                // Counter delta with 32-bit wrap support.
                // This also allows negative movement when converted to DINT.
                counterDeltaCh1 := UDINT_TO_DINT(encoderPositionRawValue - lastCounterValueCh1);

                // Convert pulses to millimeters
                positionDeltaCh1 := DINT_TO_REAL(counterDeltaCh1) * encoderScalingFactor;

                // Calculate speed
                channel1EncoderSpeedMMs := positionDeltaCh1 / calculationTimeSec;
                channel1EncoderSpeedMPM := channel1EncoderSpeedMMs * 60.0 / 1000.0;

                // Absolute speed
                channel1EncoderSpeedAbsMMs := ABS(channel1EncoderSpeedMMs);
                channel1EncoderSpeedAbsMPM := ABS(channel1EncoderSpeedMPM);

            ELSE
                // First cycle has no valid previous counter
                channel1EncoderSpeedMMs    := 0.0;
                channel1EncoderSpeedMPM    := 0.0;
                channel1EncoderSpeedAbsMMs := 0.0;
                channel1EncoderSpeedAbsMPM := 0.0;

                firstCycleCh1 := FALSE;
            END_IF

            // Store current counter for next calculation
            lastCounterValueCh1 := encoderPositionRawValue;
        END_IF


    //==============================================================
    // CHANNEL 2
    //==============================================================
    2:
        instTON_calculateEncSpeedCh2(IN := TRUE, PT := speedCalculationCycleTime);

        IF instTON_calculateEncSpeedCh2.Q THEN
            // Reset timer
            instTON_calculateEncSpeedCh2(IN := FALSE);

            IF NOT firstCycleCh2 THEN

                // Counter delta with 32-bit wrap support.
                // This also allows negative movement when converted to DINT.
                counterDeltaCh2 := UDINT_TO_DINT(encoderPositionRawValue - lastCounterValueCh2);

                // Convert pulses to millimeters
                positionDeltaCh2 := DINT_TO_REAL(counterDeltaCh2) * encoderScalingFactor;

                // Calculate speed
                channel2EncoderSpeedMMs := positionDeltaCh2 / calculationTimeSec;
                channel2EncoderSpeedMPM := channel2EncoderSpeedMMs * 60.0 / 1000.0;

                // Absolute speed
                channel2EncoderSpeedAbsMMs := ABS(channel2EncoderSpeedMMs);
                channel2EncoderSpeedAbsMPM := ABS(channel2EncoderSpeedMPM);

            ELSE
                // First cycle has no valid previous counter
                channel2EncoderSpeedMMs    := 0.0;
                channel2EncoderSpeedMPM    := 0.0;
                channel2EncoderSpeedAbsMMs := 0.0;
                channel2EncoderSpeedAbsMPM := 0.0;

                firstCycleCh2 := FALSE;
            END_IF

            // Store current counter for next calculation
            lastCounterValueCh2 := encoderPositionRawValue;
        END_IF

END_CASE
END_METHOD

METHOD PRIVATE _CalculateModuloPosition : LREAL
// ==================================================================================================
// Calculates modulo position without using FLOOR.
//
// Output range:
//   0.0 <= modulo position < moduloPosition
//
// Example:
//   absolutePosition = 725.0
//   moduloPosition   = 360.0
//   return           = 5.0
// ==================================================================================================

VAR_INPUT
    absolutePosition : LREAL; // Absolute accumulated position
    moduloPosition   : LREAL; // Modulo range, for example 360.0
END_VAR

VAR
    quotient    : LINT;
    moduloValue : LREAL;
END_VAR


// If modulo is disabled or invalid, return absolute position
IF moduloPosition <= 0.0 THEN
    _CalculateModuloPosition := absolutePosition;
    RETURN;
END_IF


// Approximate quotient.
// Depending on the PLC/runtime, LREAL_TO_LINT may truncate or round.
// The correction below guarantees the final value stays inside the modulo range.
quotient := LREAL_TO_LINT(absolutePosition / moduloPosition);


// Calculate initial modulo value
moduloValue := absolutePosition - (LINT_TO_LREAL(quotient) * moduloPosition);


// Correct negative residue
WHILE moduloValue < 0.0 DO
    moduloValue := moduloValue + moduloPosition;
END_WHILE


// Correct value above modulo range
WHILE moduloValue >= moduloPosition DO
    moduloValue := moduloValue - moduloPosition;
END_WHILE


_CalculateModuloPosition := moduloValue;
END_METHOD

METHOD PRIVATE _SetEncoderPosition
// ==================================================================================================
// Sets encoder position for channel 1 or channel 2.
//
// The command is triggered on the rising edge of setPosition.
// The desired position in millimeters is converted to raw encoder pulses.
// ==================================================================================================

VAR_INPUT
    channel              : USINT; // 1 = Channel 1, 2 = Channel 2
    setPosition          : BOOL;  // Rising edge command
    desiredPosition      : LREAL; // Desired position in mm
    encoderScalingFactor : REAL;  // mm per pulse
END_VAR

VAR
    setPositionRawValue : UDINT;
END_VAR


IF encoderScalingFactor <= 0.0 THEN
    RETURN;
END_IF


// Convert desired position from mm to raw encoder pulses
setPositionRawValue := LREAL_TO_UDINT(desiredPosition / REAL_TO_LREAL(encoderScalingFactor));


CASE channel OF

    //==============================================================
    // CHANNEL 1
    //==============================================================
    1:

        // Rising edge detection
        IF setPosition AND NOT channel1SetPositionOld THEN

            channel1SetPositionRawValue := setPositionRawValue;

            // Write raw set value to output PDO
            // Adjust these member names according to your EL5152_PLCTOHW structure
            PlcToHw.channel1.setCounterValue := channel1SetPositionRawValue;

            // Generate one PLC-cycle command pulse
            // Adjust this member name according to your EL5152_PLCTOHW structure
            PlcToHw.channel1.control.Set_counter := TRUE;

            // Avoid false speed spike after position jump
            firstCycleCh1 := TRUE;

        ELSE

            // Reset command bit after one PLC cycle
            // Adjust this member name according to your EL5152_PLCTOHW structure
            PlcToHw.channel1.control.Set_counter := FALSE;

        END_IF

        channel1SetPositionOld := setPosition;


    //==============================================================
    // CHANNEL 2
    //==============================================================
    2:

        // Rising edge detection
        IF setPosition AND NOT channel2SetPositionOld THEN

            channel2SetPositionRawValue := setPositionRawValue;

            // Write raw set value to output PDO
            // Adjust these member names according to your EL5152_PLCTOHW structure
            PlcToHw.channel2.setCounterValue := channel2SetPositionRawValue;

            // Generate one PLC-cycle command pulse
            // Adjust this member name according to your EL5152_PLCTOHW structure
            PlcToHw.channel2.control.Set_counter := TRUE;

            // Avoid false speed spike after position jump
            firstCycleCh2 := TRUE;

        ELSE

            // Reset command bit after one PLC cycle
            // Adjust this member name according to your EL5152_PLCTOHW structure
            PlcToHw.channel2.control.Set_counter := FALSE;

        END_IF

        channel2SetPositionOld := setPosition;

END_CASE
END_METHOD

METHOD PRIVATE _SimulateEncoderSpeed : UDINT
// ==================================================================================================
// Simulates encoder motion by incrementing a virtual counter value based on a given speed in m/min.
//
// Positive simulateSpeedMPM increases the raw counter.
// Negative simulateSpeedMPM decreases the raw counter.
// ==================================================================================================

VAR_INPUT
    channel              : USINT; // 1 = Channel 1, 2 = Channel 2
    encoderScalingFactor : REAL;  // Encoder resolution: mm per pulse
    simulateSpeedMPM     : REAL;  // Target speed in meters per minute
END_VAR


IF encoderScalingFactor <= 0.0 THEN
    RETURN;
END_IF


CASE channel OF

    //==============================================================
    // CHANNEL 1
    //==============================================================
    1:
        currentSystemTimeCh1 := F_GetSystemTime();

        // Initialize simulation time reference
        IF NOT simulationInitCh1 THEN
            lastCycleTimeCh1 := currentSystemTimeCh1;
            simulationInitCh1 := TRUE;
            _SimulateEncoderSpeed := simulatedPositionRawValueCh1;
            RETURN;
        END_IF

        // 1 tick = 100 ns
        // 1 ms = 10,000 ticks
        deltaTimeMsCh1 := ULINT_TO_REAL(currentSystemTimeCh1 - lastCycleTimeCh1) / 10000.0;

        // Store time for next cycle
        lastCycleTimeCh1 := currentSystemTimeCh1;

        IF deltaTimeMsCh1 > 0.0 THEN

            // Convert m/min to pulses per second
            pulsesPerSecondCh1 := (simulateSpeedMPM * 1000.0 / 60.0) / encoderScalingFactor;

            // Convert pulses per second to pulses per cycle
            pulsesToAddCh1 := REAL_TO_DINT(pulsesPerSecondCh1 * (deltaTimeMsCh1 / 1000.0));

            IF pulsesToAddCh1 >= 0 THEN
                simulatedPositionRawValueCh1 := simulatedPositionRawValueCh1 + DINT_TO_UDINT(pulsesToAddCh1);
            ELSE
                simulatedPositionRawValueCh1 := simulatedPositionRawValueCh1 - DINT_TO_UDINT(ABS(pulsesToAddCh1));
            END_IF

        END_IF

        _SimulateEncoderSpeed := simulatedPositionRawValueCh1;


    //==============================================================
    // CHANNEL 2
    //==============================================================
    2:
        currentSystemTimeCh2 := F_GetSystemTime();

        // Initialize simulation time reference
        IF NOT simulationInitCh2 THEN
            lastCycleTimeCh2 := currentSystemTimeCh2;
            simulationInitCh2 := TRUE;
            _SimulateEncoderSpeed := simulatedPositionRawValueCh2;
            RETURN;
        END_IF

        // 1 tick = 100 ns
        // 1 ms = 10,000 ticks
        deltaTimeMsCh2 := ULINT_TO_REAL(currentSystemTimeCh2 - lastCycleTimeCh2) / 10000.0;

        // Store time for next cycle
        lastCycleTimeCh2 := currentSystemTimeCh2;

        IF deltaTimeMsCh2 > 0.0 THEN

            // Convert m/min to pulses per second
            pulsesPerSecondCh2 := (simulateSpeedMPM * 1000.0 / 60.0) / encoderScalingFactor;

            // Convert pulses per second to pulses per cycle
            pulsesToAddCh2 := REAL_TO_DINT(pulsesPerSecondCh2 * (deltaTimeMsCh2 / 1000.0));

            IF pulsesToAddCh2 >= 0 THEN
                simulatedPositionRawValueCh2 := simulatedPositionRawValueCh2 + DINT_TO_UDINT(pulsesToAddCh2);
            ELSE
                simulatedPositionRawValueCh2 := simulatedPositionRawValueCh2 - DINT_TO_UDINT(ABS(pulsesToAddCh2));
            END_IF

        END_IF

        _SimulateEncoderSpeed := simulatedPositionRawValueCh2;

END_CASE
END_METHOD

END_FUNCTION_BLOCK

// ---- Library/FAS/IO-Link/006B51 - IO-Link Master/_FB_006B51.TcPOU
FUNCTION_BLOCK _FB_006B51
VAR_INPUT
	
		
END_VAR
VAR_OUTPUT
	
	channel_0 : _006B51_Channel_State;
	channel_1 : _006B51_Channel_State;
	channel_2 : _006B51_Channel_State;
	channel_3 : _006B51_Channel_State;
	channel_4 : _006B51_Channel_State;
	channel_5 : _006B51_Channel_State;
	channel_6 : _006B51_Channel_State;
	channel_7 : _006B51_Channel_State;
	
	HwToPlc	AT %I* 	: _006B51_HWTOPLC_PDOS;	
			
END_VAR

//============================================================
// CHANNEL 0
//============================================================
channel_0.inputPin2   := HwToPlc.inputPin2.00;
channel_0.inputPin4   := HwToPlc.inputPin4.00;
channel_0.deviceState := HwToPlc.deviceState.00;

// Reset port mode states
channel_0.state_PortInNoDigitalInput        := FALSE;
channel_0.state_PortInNcDigitalInput        := FALSE;
channel_0.state_PortInDigitalOutput         := FALSE;
channel_0.state_PortInIoLink                := FALSE;

// Reset diagnostic / communication states
channel_0.state_NoDeviceDetected            := FALSE;
channel_0.state_IoLinkCommunicationStatus   := FALSE;
channel_0.state_InvalidVendorId             := FALSE;
channel_0.state_InvalidDeviceId             := FALSE;
channel_0.state_InvalidSerialNumber         := FALSE;
channel_0.state_InvalidCycleTime            := FALSE;
channel_0.state_InvalidProcessDataInLength  := FALSE;
channel_0.state_InvalidProcessDataOutLength := FALSE;
channel_0.state_InvalidIoLinkVersion        := FALSE;

// Low nibble = port mode
CASE (HwToPlc.ioLinkDeviceState_Port0 AND 16#0F) OF
    16#0: channel_0.state_PortInNoDigitalInput := TRUE;
    16#1: channel_0.state_PortInNcDigitalInput := TRUE;
    16#2: channel_0.state_PortInDigitalOutput  := TRUE;
    16#3: channel_0.state_PortInIoLink         := TRUE;
END_CASE;

// High nibble = diagnostic / communication state
CASE SHR((HwToPlc.ioLinkDeviceState_Port0 AND 16#F0), 4) OF
    16#0: channel_0.state_NoDeviceDetected            := TRUE;
    16#1: channel_0.state_IoLinkCommunicationStatus   := TRUE;
    16#2: channel_0.state_InvalidVendorId             := TRUE;
    16#3: channel_0.state_InvalidDeviceId             := TRUE;
    16#4: channel_0.state_InvalidSerialNumber         := TRUE;
    16#8: channel_0.state_InvalidCycleTime            := TRUE;
    16#9: channel_0.state_InvalidProcessDataInLength  := TRUE;
    16#A: channel_0.state_InvalidProcessDataOutLength := TRUE;
    16#C: channel_0.state_InvalidIoLinkVersion        := TRUE;
END_CASE;


//============================================================
// CHANNEL 1
//============================================================
channel_1.inputPin2   := HwToPlc.inputPin2.01;
channel_1.inputPin4   := HwToPlc.inputPin4.01;
channel_1.deviceState := HwToPlc.deviceState.01;

// Reset port mode states
channel_1.state_PortInNoDigitalInput        := FALSE;
channel_1.state_PortInNcDigitalInput        := FALSE;
channel_1.state_PortInDigitalOutput         := FALSE;
channel_1.state_PortInIoLink                := FALSE;

// Reset diagnostic / communication states
channel_1.state_NoDeviceDetected            := FALSE;
channel_1.state_IoLinkCommunicationStatus   := FALSE;
channel_1.state_InvalidVendorId             := FALSE;
channel_1.state_InvalidDeviceId             := FALSE;
channel_1.state_InvalidSerialNumber         := FALSE;
channel_1.state_InvalidCycleTime            := FALSE;
channel_1.state_InvalidProcessDataInLength  := FALSE;
channel_1.state_InvalidProcessDataOutLength := FALSE;
channel_1.state_InvalidIoLinkVersion        := FALSE;

// Low nibble = port mode
CASE (HwToPlc.ioLinkDeviceState_Port1 AND 16#0F) OF
    16#0: channel_1.state_PortInNoDigitalInput := TRUE;
    16#1: channel_1.state_PortInNcDigitalInput := TRUE;
    16#2: channel_1.state_PortInDigitalOutput  := TRUE;
    16#3: channel_1.state_PortInIoLink         := TRUE;
END_CASE;

// High nibble = diagnostic / communication state
CASE SHR((HwToPlc.ioLinkDeviceState_Port1 AND 16#F0), 4) OF
    16#0: channel_1.state_NoDeviceDetected            := TRUE;
    16#1: channel_1.state_IoLinkCommunicationStatus   := TRUE;
    16#2: channel_1.state_InvalidVendorId             := TRUE;
    16#3: channel_1.state_InvalidDeviceId             := TRUE;
    16#4: channel_1.state_InvalidSerialNumber         := TRUE;
    16#8: channel_1.state_InvalidCycleTime            := TRUE;
    16#9: channel_1.state_InvalidProcessDataInLength  := TRUE;
    16#A: channel_1.state_InvalidProcessDataOutLength := TRUE;
    16#C: channel_1.state_InvalidIoLinkVersion        := TRUE;
END_CASE;


//============================================================
// CHANNEL 2
//============================================================
channel_2.inputPin2   := HwToPlc.inputPin2.02;
channel_2.inputPin4   := HwToPlc.inputPin4.02;
channel_2.deviceState := HwToPlc.deviceState.02;

// Reset port mode states
channel_2.state_PortInNoDigitalInput        := FALSE;
channel_2.state_PortInNcDigitalInput        := FALSE;
channel_2.state_PortInDigitalOutput         := FALSE;
channel_2.state_PortInIoLink                := FALSE;

// Reset diagnostic / communication states
channel_2.state_NoDeviceDetected            := FALSE;
channel_2.state_IoLinkCommunicationStatus   := FALSE;
channel_2.state_InvalidVendorId             := FALSE;
channel_2.state_InvalidDeviceId             := FALSE;
channel_2.state_InvalidSerialNumber         := FALSE;
channel_2.state_InvalidCycleTime            := FALSE;
channel_2.state_InvalidProcessDataInLength  := FALSE;
channel_2.state_InvalidProcessDataOutLength := FALSE;
channel_2.state_InvalidIoLinkVersion        := FALSE;

// Low nibble = port mode
CASE (HwToPlc.ioLinkDeviceState_Port2 AND 16#0F) OF
    16#0: channel_2.state_PortInNoDigitalInput := TRUE;
    16#1: channel_2.state_PortInNcDigitalInput := TRUE;
    16#2: channel_2.state_PortInDigitalOutput  := TRUE;
    16#3: channel_2.state_PortInIoLink         := TRUE;
END_CASE;

// High nibble = diagnostic / communication state
CASE SHR((HwToPlc.ioLinkDeviceState_Port2 AND 16#F0), 4) OF
    16#0: channel_2.state_NoDeviceDetected            := TRUE;
    16#1: channel_2.state_IoLinkCommunicationStatus   := TRUE;
    16#2: channel_2.state_InvalidVendorId             := TRUE;
    16#3: channel_2.state_InvalidDeviceId             := TRUE;
    16#4: channel_2.state_InvalidSerialNumber         := TRUE;
    16#8: channel_2.state_InvalidCycleTime            := TRUE;
    16#9: channel_2.state_InvalidProcessDataInLength  := TRUE;
    16#A: channel_2.state_InvalidProcessDataOutLength := TRUE;
    16#C: channel_2.state_InvalidIoLinkVersion        := TRUE;
END_CASE;


//============================================================
// CHANNEL 3
//============================================================
channel_3.inputPin2   := HwToPlc.inputPin2.03;
channel_3.inputPin4   := HwToPlc.inputPin4.03;
channel_3.deviceState := HwToPlc.deviceState.03;

// Reset port mode states
channel_3.state_PortInNoDigitalInput        := FALSE;
channel_3.state_PortInNcDigitalInput        := FALSE;
channel_3.state_PortInDigitalOutput         := FALSE;
channel_3.state_PortInIoLink                := FALSE;

// Reset diagnostic / communication states
channel_3.state_NoDeviceDetected            := FALSE;
channel_3.state_IoLinkCommunicationStatus   := FALSE;
channel_3.state_InvalidVendorId             := FALSE;
channel_3.state_InvalidDeviceId             := FALSE;
channel_3.state_InvalidSerialNumber         := FALSE;
channel_3.state_InvalidCycleTime            := FALSE;
channel_3.state_InvalidProcessDataInLength  := FALSE;
channel_3.state_InvalidProcessDataOutLength := FALSE;
channel_3.state_InvalidIoLinkVersion        := FALSE;

// Low nibble = port mode
CASE (HwToPlc.ioLinkDeviceState_Port3 AND 16#0F) OF
    16#0: channel_3.state_PortInNoDigitalInput := TRUE;
    16#1: channel_3.state_PortInNcDigitalInput := TRUE;
    16#2: channel_3.state_PortInDigitalOutput  := TRUE;
    16#3: channel_3.state_PortInIoLink         := TRUE;
END_CASE;

// High nibble = diagnostic / communication state
CASE SHR((HwToPlc.ioLinkDeviceState_Port3 AND 16#F0), 4) OF
    16#0: channel_3.state_NoDeviceDetected            := TRUE;
    16#1: channel_3.state_IoLinkCommunicationStatus   := TRUE;
    16#2: channel_3.state_InvalidVendorId             := TRUE;
    16#3: channel_3.state_InvalidDeviceId             := TRUE;
    16#4: channel_3.state_InvalidSerialNumber         := TRUE;
    16#8: channel_3.state_InvalidCycleTime            := TRUE;
    16#9: channel_3.state_InvalidProcessDataInLength  := TRUE;
    16#A: channel_3.state_InvalidProcessDataOutLength := TRUE;
    16#C: channel_3.state_InvalidIoLinkVersion        := TRUE;
END_CASE;


//============================================================
// CHANNEL 4
//============================================================
channel_4.inputPin2   := HwToPlc.inputPin2.04;
channel_4.inputPin4   := HwToPlc.inputPin4.04;
channel_4.deviceState := HwToPlc.deviceState.04;

// Reset port mode states
channel_4.state_PortInNoDigitalInput        := FALSE;
channel_4.state_PortInNcDigitalInput        := FALSE;
channel_4.state_PortInDigitalOutput         := FALSE;
channel_4.state_PortInIoLink                := FALSE;

// Reset diagnostic / communication states
channel_4.state_NoDeviceDetected            := FALSE;
channel_4.state_IoLinkCommunicationStatus   := FALSE;
channel_4.state_InvalidVendorId             := FALSE;
channel_4.state_InvalidDeviceId             := FALSE;
channel_4.state_InvalidSerialNumber         := FALSE;
channel_4.state_InvalidCycleTime            := FALSE;
channel_4.state_InvalidProcessDataInLength  := FALSE;
channel_4.state_InvalidProcessDataOutLength := FALSE;
channel_4.state_InvalidIoLinkVersion        := FALSE;

// Low nibble = port mode
CASE (HwToPlc.ioLinkDeviceState_Port4 AND 16#0F) OF
    16#0: channel_4.state_PortInNoDigitalInput := TRUE;
    16#1: channel_4.state_PortInNcDigitalInput := TRUE;
    16#2: channel_4.state_PortInDigitalOutput  := TRUE;
    16#3: channel_4.state_PortInIoLink         := TRUE;
END_CASE;

// High nibble = diagnostic / communication state
CASE SHR((HwToPlc.ioLinkDeviceState_Port4 AND 16#F0), 4) OF
    16#0: channel_4.state_NoDeviceDetected            := TRUE;
    16#1: channel_4.state_IoLinkCommunicationStatus   := TRUE;
    16#2: channel_4.state_InvalidVendorId             := TRUE;
    16#3: channel_4.state_InvalidDeviceId             := TRUE;
    16#4: channel_4.state_InvalidSerialNumber         := TRUE;
    16#8: channel_4.state_InvalidCycleTime            := TRUE;
    16#9: channel_4.state_InvalidProcessDataInLength  := TRUE;
    16#A: channel_4.state_InvalidProcessDataOutLength := TRUE;
    16#C: channel_4.state_InvalidIoLinkVersion        := TRUE;
END_CASE;


//============================================================
// CHANNEL 5
//============================================================
channel_5.inputPin2   := HwToPlc.inputPin2.05;
channel_5.inputPin4   := HwToPlc.inputPin4.05;
channel_5.deviceState := HwToPlc.deviceState.05;

// Reset port mode states
channel_5.state_PortInNoDigitalInput        := FALSE;
channel_5.state_PortInNcDigitalInput        := FALSE;
channel_5.state_PortInDigitalOutput         := FALSE;
channel_5.state_PortInIoLink                := FALSE;

// Reset diagnostic / communication states
channel_5.state_NoDeviceDetected            := FALSE;
channel_5.state_IoLinkCommunicationStatus   := FALSE;
channel_5.state_InvalidVendorId             := FALSE;
channel_5.state_InvalidDeviceId             := FALSE;
channel_5.state_InvalidSerialNumber         := FALSE;
channel_5.state_InvalidCycleTime            := FALSE;
channel_5.state_InvalidProcessDataInLength  := FALSE;
channel_5.state_InvalidProcessDataOutLength := FALSE;
channel_5.state_InvalidIoLinkVersion        := FALSE;

// Low nibble = port mode
CASE (HwToPlc.ioLinkDeviceState_Port5 AND 16#0F) OF
    16#0: channel_5.state_PortInNoDigitalInput := TRUE;
    16#1: channel_5.state_PortInNcDigitalInput := TRUE;
    16#2: channel_5.state_PortInDigitalOutput  := TRUE;
    16#3: channel_5.state_PortInIoLink         := TRUE;
END_CASE;

// High nibble = diagnostic / communication state
CASE SHR((HwToPlc.ioLinkDeviceState_Port5 AND 16#F0), 4) OF
    16#0: channel_5.state_NoDeviceDetected            := TRUE;
    16#1: channel_5.state_IoLinkCommunicationStatus   := TRUE;
    16#2: channel_5.state_InvalidVendorId             := TRUE;
    16#3: channel_5.state_InvalidDeviceId             := TRUE;
    16#4: channel_5.state_InvalidSerialNumber         := TRUE;
    16#8: channel_5.state_InvalidCycleTime            := TRUE;
    16#9: channel_5.state_InvalidProcessDataInLength  := TRUE;
    16#A: channel_5.state_InvalidProcessDataOutLength := TRUE;
    16#C: channel_5.state_InvalidIoLinkVersion        := TRUE;
END_CASE;


//============================================================
// CHANNEL 6
//============================================================
channel_6.inputPin2   := HwToPlc.inputPin2.06;
channel_6.inputPin4   := HwToPlc.inputPin4.06;
channel_6.deviceState := HwToPlc.deviceState.06;

// Reset port mode states
channel_6.state_PortInNoDigitalInput        := FALSE;
channel_6.state_PortInNcDigitalInput        := FALSE;
channel_6.state_PortInDigitalOutput         := FALSE;
channel_6.state_PortInIoLink                := FALSE;

// Reset diagnostic / communication states
channel_6.state_NoDeviceDetected            := FALSE;
channel_6.state_IoLinkCommunicationStatus   := FALSE;
channel_6.state_InvalidVendorId             := FALSE;
channel_6.state_InvalidDeviceId             := FALSE;
channel_6.state_InvalidSerialNumber         := FALSE;
channel_6.state_InvalidCycleTime            := FALSE;
channel_6.state_InvalidProcessDataInLength  := FALSE;
channel_6.state_InvalidProcessDataOutLength := FALSE;
channel_6.state_InvalidIoLinkVersion        := FALSE;

// Low nibble = port mode
CASE (HwToPlc.ioLinkDeviceState_Port6 AND 16#0F) OF
    16#0: channel_6.state_PortInNoDigitalInput := TRUE;
    16#1: channel_6.state_PortInNcDigitalInput := TRUE;
    16#2: channel_6.state_PortInDigitalOutput  := TRUE;
    16#3: channel_6.state_PortInIoLink         := TRUE;
END_CASE;

// High nibble = diagnostic / communication state
CASE SHR((HwToPlc.ioLinkDeviceState_Port6 AND 16#F0), 4) OF
    16#0: channel_6.state_NoDeviceDetected            := TRUE;
    16#1: channel_6.state_IoLinkCommunicationStatus   := TRUE;
    16#2: channel_6.state_InvalidVendorId             := TRUE;
    16#3: channel_6.state_InvalidDeviceId             := TRUE;
    16#4: channel_6.state_InvalidSerialNumber         := TRUE;
    16#8: channel_6.state_InvalidCycleTime            := TRUE;
    16#9: channel_6.state_InvalidProcessDataInLength  := TRUE;
    16#A: channel_6.state_InvalidProcessDataOutLength := TRUE;
    16#C: channel_6.state_InvalidIoLinkVersion        := TRUE;
END_CASE;


//============================================================
// CHANNEL 7
//============================================================
channel_7.inputPin2   := HwToPlc.inputPin2.07;
channel_7.inputPin4   := HwToPlc.inputPin4.07;
channel_7.deviceState := HwToPlc.deviceState.07;

// Reset port mode states
channel_7.state_PortInNoDigitalInput        := FALSE;
channel_7.state_PortInNcDigitalInput        := FALSE;
channel_7.state_PortInDigitalOutput         := FALSE;
channel_7.state_PortInIoLink                := FALSE;

// Reset diagnostic / communication states
channel_7.state_NoDeviceDetected            := FALSE;
channel_7.state_IoLinkCommunicationStatus   := FALSE;
channel_7.state_InvalidVendorId             := FALSE;
channel_7.state_InvalidDeviceId             := FALSE;
channel_7.state_InvalidSerialNumber         := FALSE;
channel_7.state_InvalidCycleTime            := FALSE;
channel_7.state_InvalidProcessDataInLength  := FALSE;
channel_7.state_InvalidProcessDataOutLength := FALSE;
channel_7.state_InvalidIoLinkVersion        := FALSE;

// Low nibble = port mode
CASE (HwToPlc.ioLinkDeviceState_Port7 AND 16#0F) OF
    16#0: channel_7.state_PortInNoDigitalInput := TRUE;
    16#1: channel_7.state_PortInNcDigitalInput := TRUE;
    16#2: channel_7.state_PortInDigitalOutput  := TRUE;
    16#3: channel_7.state_PortInIoLink         := TRUE;
END_CASE;

// High nibble = diagnostic / communication state
CASE SHR((HwToPlc.ioLinkDeviceState_Port7 AND 16#F0), 4) OF
    16#0: channel_7.state_NoDeviceDetected            := TRUE;
    16#1: channel_7.state_IoLinkCommunicationStatus   := TRUE;
    16#2: channel_7.state_InvalidVendorId             := TRUE;
    16#3: channel_7.state_InvalidDeviceId             := TRUE;
    16#4: channel_7.state_InvalidSerialNumber         := TRUE;
    16#8: channel_7.state_InvalidCycleTime            := TRUE;
    16#9: channel_7.state_InvalidProcessDataInLength  := TRUE;
    16#A: channel_7.state_InvalidProcessDataOutLength := TRUE;
    16#C: channel_7.state_InvalidIoLinkVersion        := TRUE;
END_CASE;

END_FUNCTION_BLOCK

// ---- Library/FAS/IO-Link/00BE31 - IP67 16Di or 16Do/_FB_00BE31.TcPOU
FUNCTION_BLOCK _FB_00BE31
VAR_INPUT
	
	ch0_Output_Pin2 : BOOL;
	ch0_Output_Pin4 : BOOL;	
	ch1_Output_Pin2 : BOOL;
	ch1_Output_Pin4 : BOOL;	
	ch2_Output_Pin2 : BOOL;
	ch2_Output_Pin4 : BOOL;		
	ch3_Output_Pin2 : BOOL;
	ch3_Output_Pin4 : BOOL;	
	ch4_Output_Pin2 : BOOL;
	ch4_Output_Pin4 : BOOL;		
	ch5_Output_Pin2 : BOOL;
	ch5_Output_Pin4 : BOOL;			
	ch6_Output_Pin2 : BOOL;
	ch6_Output_Pin4 : BOOL;		
	ch7_Output_Pin2 : BOOL;
	ch7_Output_Pin4 : BOOL;		
	
	PlcToHw	AT %Q* 	: _00BE31_PLCTOHW_PDOS;	
		
END_VAR
VAR_OUTPUT
	
	ch0_Input_Pin2 : BOOL;
	ch0_Input_Pin4 : BOOL;	
	ch1_Input_Pin2 : BOOL;
	ch1_Input_Pin4 : BOOL;
	ch2_Input_Pin2 : BOOL;
	ch2_Input_Pin4 : BOOL;
	ch3_Input_Pin2 : BOOL;
	ch3_Input_Pin4 : BOOL;	
	ch4_Input_Pin2 : BOOL;
	ch4_Input_Pin4 : BOOL;	
	ch5_Input_Pin2 : BOOL;
	ch5_Input_Pin4 : BOOL;		
	ch6_Input_Pin2 : BOOL;
	ch6_Input_Pin4 : BOOL;	
	ch7_Input_Pin2 : BOOL;
	ch7_Input_Pin4 : BOOL;
	
	HwToPlc	AT %I* 	: _00BE31_HWTOPLC_PDOS;	
	
			
END_VAR
VAR


END_VAR

PlcToHw.outputByte_1.0 := ch0_Output_Pin2;
PlcToHw.outputByte_0.0 := ch0_Output_Pin4;

PlcToHw.outputByte_1.1 := ch1_Output_Pin2;
PlcToHw.outputByte_0.1 := ch1_Output_Pin4;

PlcToHw.outputByte_1.2 := ch2_Output_Pin2;
PlcToHw.outputByte_0.2 := ch2_Output_Pin4;

PlcToHw.outputByte_1.3 := ch3_Output_Pin2;
PlcToHw.outputByte_0.3 := ch3_Output_Pin4;

PlcToHw.outputByte_1.4 := ch4_Output_Pin2;
PlcToHw.outputByte_0.4 := ch4_Output_Pin4;

PlcToHw.outputByte_1.5 := ch5_Output_Pin2;
PlcToHw.outputByte_0.5 := ch5_Output_Pin4;

PlcToHw.outputByte_1.6 := ch6_Output_Pin2;
PlcToHw.outputByte_0.6 := ch6_Output_Pin4;

PlcToHw.outputByte_1.7 := ch7_Output_Pin2;
PlcToHw.outputByte_0.7 := ch7_Output_Pin4;


ch0_Input_Pin2 := HwToPlc.inputByte_1.0;
ch0_Input_Pin4 := HwToPlc.inputByte_0.0;

ch1_Input_Pin2 := HwToPlc.inputByte_1.1;
ch1_Input_Pin4 := HwToPlc.inputByte_0.1;

ch2_Input_Pin2 := HwToPlc.inputByte_1.2;
ch2_Input_Pin4 := HwToPlc.inputByte_0.2;

ch3_Input_Pin2 := HwToPlc.inputByte_1.3;
ch3_Input_Pin4 := HwToPlc.inputByte_0.3;

ch4_Input_Pin2 := HwToPlc.inputByte_1.4;
ch4_Input_Pin4 := HwToPlc.inputByte_0.4;

ch5_Input_Pin2 := HwToPlc.inputByte_1.5;
ch5_Input_Pin4 := HwToPlc.inputByte_0.5;

ch6_Input_Pin2 := HwToPlc.inputByte_1.6;
ch6_Input_Pin4 := HwToPlc.inputByte_0.6;

ch7_Input_Pin2 := HwToPlc.inputByte_1.7;
ch7_Input_Pin4 := HwToPlc.inputByte_0.7;

END_FUNCTION_BLOCK

// ---- Library/FAS/IO-Link/00BH11 - 16Di or 16Do/_FB_00BH11.TcPOU
FUNCTION_BLOCK _FB_00BH11
VAR_INPUT
	
	digitalOutput_01 : BOOL;
	digitalOutput_02 : BOOL;
	digitalOutput_03 : BOOL;
	digitalOutput_04 : BOOL;
	digitalOutput_05 : BOOL;
	digitalOutput_06 : BOOL;
	digitalOutput_07 : BOOL;
	digitalOutput_08 : BOOL;
	digitalOutput_09 : BOOL;
	digitalOutput_10 : BOOL;
	digitalOutput_11 : BOOL;
	digitalOutput_12 : BOOL;
	digitalOutput_13 : BOOL;
	digitalOutput_14 : BOOL;
	digitalOutput_15 : BOOL;
	digitalOutput_16 : BOOL;
	
	PlcToHw	AT %Q* 	: _00BH11_PLCTOHW_PDOS;	
		
END_VAR
VAR_OUTPUT
	
	digitalInput_01  : BOOL;
	digitalInput_02  : BOOL;
	digitalInput_03  : BOOL;
	digitalInput_04  : BOOL;
	digitalInput_05  : BOOL;
	digitalInput_06  : BOOL;
	digitalInput_07  : BOOL;
	digitalInput_08  : BOOL;
	digitalInput_09  : BOOL;
	digitalInput_10  : BOOL;
	digitalInput_11  : BOOL;
	digitalInput_12  : BOOL;
	digitalInput_13  : BOOL;
	digitalInput_14  : BOOL;
	digitalInput_15  : BOOL;
	digitalInput_16  : BOOL;
	
	
	HwToPlc	AT %I* 	: _00BH11_HWTOPLC_PDOS;	
	
			
END_VAR
VAR


END_VAR

//==============================================================
// Digital Inputs
//==============================================================

digitalInput_01 := HwToPlc.inputByte_0.0;
digitalInput_02 := HwToPlc.inputByte_0.1;
digitalInput_03 := HwToPlc.inputByte_0.2;
digitalInput_04 := HwToPlc.inputByte_0.3;
digitalInput_05 := HwToPlc.inputByte_0.4;
digitalInput_06 := HwToPlc.inputByte_0.5;
digitalInput_07 := HwToPlc.inputByte_0.6;
digitalInput_08 := HwToPlc.inputByte_0.7;

digitalInput_09 := HwToPlc.inputByte_1.0;
digitalInput_10 := HwToPlc.inputByte_1.1;
digitalInput_11 := HwToPlc.inputByte_1.2;
digitalInput_12 := HwToPlc.inputByte_1.3;
digitalInput_13 := HwToPlc.inputByte_1.4;
digitalInput_14 := HwToPlc.inputByte_1.5;
digitalInput_15 := HwToPlc.inputByte_1.6;
digitalInput_16 := HwToPlc.inputByte_1.7;


//==============================================================
// Digital Outputs
//==============================================================

PlcToHw.outputByte_0.0 := digitalOutput_01;
PlcToHw.outputByte_0.1 := digitalOutput_02;
PlcToHw.outputByte_0.2 := digitalOutput_03;
PlcToHw.outputByte_0.3 := digitalOutput_04;
PlcToHw.outputByte_0.4 := digitalOutput_05;
PlcToHw.outputByte_0.5 := digitalOutput_06;
PlcToHw.outputByte_0.6 := digitalOutput_07;
PlcToHw.outputByte_0.7 := digitalOutput_08;

PlcToHw.outputByte_1.0 := digitalOutput_09;
PlcToHw.outputByte_1.1 := digitalOutput_10;
PlcToHw.outputByte_1.2 := digitalOutput_11;
PlcToHw.outputByte_1.3 := digitalOutput_12;
PlcToHw.outputByte_1.4 := digitalOutput_13;
PlcToHw.outputByte_1.5 := digitalOutput_14;
PlcToHw.outputByte_1.6 := digitalOutput_15;
PlcToHw.outputByte_1.7 := digitalOutput_16;

END_FUNCTION_BLOCK

// ---- Library/Sick/DT35-B15251 - Laser Sensor/_FB_DT35_B15251.TcPOU
FUNCTION_BLOCK _FB_DT35_B15251

VAR_INPUT PERSISTENT

    deviceConfig : _DT35B15251_DEV_CONFIG; // Device configuration settings

END_VAR

VAR_INPUT

    HwToPlc AT %I* : _DT35B15251_HWTOPLC_PDOS; // IO-Link input process data

END_VAR

VAR_OUTPUT

    distanceRaw      : REAL; // Raw sensor value

    distance         : REAL; // Measured distance [mm]

    distanceFromZero : REAL; // Distance relative to configured zero point [mm]

    height           : REAL; // Calculated height from reference distance [mm]

END_VAR

VAR

END_VAR




//=============================================================
// Main execution
//=============================================================

_SensorInputs();

METHOD PRIVATE _Scale : REAL
VAR_INPUT
	
	X : REAL;
	I_LO : REAL;
	I_HI : REAL;
	O_LO : REAL;
	O_HI : REAL;
	
END_VAR
IF I_LO = I_HI THEN
	_Scale := O_LO;
ELSE
	_Scale := (O_HI - O_LO) / (I_HI - I_LO) * (LIMIT(I_LO, X, I_HI) - I_LO) + O_LO;
END_IF;
END_METHOD

METHOD PRIVATE _SensorInputs
VAR
    rawDistanceWord        : WORD;
    measuredDistance       : REAL;
    calculatedDistanceZero : REAL;
    calculatedHeight       : REAL;
END_VAR

//=============================================================
// Raw sensor value
// EN: Combines the two IO-Link input bytes into one 16-bit value.
//=============================================================

rawDistanceWord := SHL(BYTE_TO_WORD(HwToPlc.inputByte_0), 8)
                   OR BYTE_TO_WORD(HwToPlc.inputByte_1);

distanceRaw := WORD_TO_REAL(rawDistanceWord);


//=============================================================
// Distance calculation
// EN: Converts process data to millimeters.
// In the default sensor configuration, the process data is already in mm.
//=============================================================

measuredDistance := distanceRaw * deviceConfig.processDataResolutionFactor;


//=============================================================
// Distance limit
// EN: Limits the measured distance to the configured valid range.
//=============================================================

distance := LIMIT(
    deviceConfig.distanceLowLimit,
    measuredDistance,
    deviceConfig.distanceHighLimit
);


//=============================================================
// Distance from zero
// EN: Calculates the distance relative to a configured zero reference.
//=============================================================

calculatedDistanceZero := distance - deviceConfig.distanceZeroReference;

distanceFromZero := LIMIT(
    deviceConfig.distanceFromZeroLowLimit,
    calculatedDistanceZero,
    deviceConfig.distanceFromZeroHighLimit
);


//=============================================================
// Height calculation
// EN: Calculates height from the measured distance.
// Higher object = smaller distance = bigger height.
//=============================================================

calculatedHeight := deviceConfig.heightReferenceDistance - distance;

height := LIMIT(
    deviceConfig.heightLowLimit,
    calculatedHeight,
    deviceConfig.heightHighLimit
);
END_METHOD

END_FUNCTION_BLOCK

// ---- Library/Inovance/IS620P-CO/FB/FB_IS620P_CO.TcPOU
FUNCTION_BLOCK FB_IS620P_CO

// =============================================================================
// EN: Generic CANopen velocity-control interface for the Inovance IS620P-CO.
//     The parent block is responsible for motion profiles, positioning logic,
//     machine limits and application safety decisions.
// PT: Interface genérica de controle de velocidade CANopen para o Inovance
//     IS620P-CO. O bloco pai é responsável pelos perfis de movimento, lógica de
//     posicionamento, limites da máquina e decisões de segurança da aplicação.
// =============================================================================

VAR_INPUT PERSISTENT
    // EN: Persistent device scaling, calibration and protection parameters.
    // PT: Parâmetros persistentes de escala, calibração e proteção do equipamento.
    deviceConfig : IS620P_CO_DEV_CONFIG;
END_VAR

VAR_INPUT
    // EN: Hardware outputs written cyclically from the PLC to the servo drive.
    // PT: Saídas de hardware escritas ciclicamente do PLC para o servo drive.
    PlcToHw AT %Q* : IS620P_CO_PLCTOHW_PDOS;

    // EN: Enables cyclic execution and output generation by this function block.
    // PT: Habilita a execução cíclica e a geração de saídas deste function block.
    enable : BOOL;

    // EN: Requests the CiA 402 Operation Enabled state.
    // PT: Solicita o estado CiA 402 Operation Enabled.
    enableDrive : BOOL;

    // EN: Rising edge requests a CiA 402 fault reset.
    // PT: A borda de subida solicita o reset de falha CiA 402.
    resetFault : BOOL;

    // EN: Requests the CiA 402 quick-stop transition with highest command priority.
    // PT: Solicita a transição de quick stop CiA 402 com maior prioridade de comando.
    quickStop : BOOL;

    // EN: Signed velocity reference generated by the parent block in millimeters per second.
    // PT: Referência de velocidade com sinal gerada pelo bloco pai em milímetros por segundo.
    velocityReferenceMmps : LREAL;

    // EN: Rising edge defines the current mechanical position as zero.
    // PT: A borda de subida define a posição mecânica atual como zero.
    zeroPosition : BOOL;

    // EN: Rising edge assigns desiredPositionMm to the current mechanical position.
    // PT: A borda de subida atribui desiredPositionMm à posição mecânica atual.
    setPosition : BOOL;

    // EN: Engineering position assigned when setPosition is triggered.
    // PT: Posição de engenharia atribuída quando setPosition é acionado.
    desiredPositionMm : LREAL;
END_VAR

VAR_OUTPUT
    // EN: Hardware inputs received cyclically from the drive and CANopen master.
    // PT: Entradas de hardware recebidas ciclicamente do drive e do mestre CANopen.
    HwToPlc AT %I* : IS620P_CO_HWTOPLC_PDOS;

    // EN: Generic communication and CiA 402 status information.
    // PT: Informações genéricas de comunicação e estado CiA 402.
    status : IS620P_CO_STATUS;

    // EN: Raw position value received from object 6064h.
    // PT: Valor bruto de posição recebido do objeto 6064h.
    rawPosition : DINT;

    // EN: Position feedback converted to millimeters before applying the offset.
    // PT: Realimentação de posição convertida para milímetros antes de aplicar o offset.
    rawPositionMm : LREAL;

    // EN: Calibrated position feedback in millimeters.
    // PT: Realimentação de posição calibrada em milímetros.
    actualPositionMm : LREAL;

    // EN: Raw velocity value received from object 606Ch.
    // PT: Valor bruto de velocidade recebido do objeto 606Ch.
    rawVelocity : DINT;

    // EN: Velocity feedback converted to millimeters per second.
    // PT: Realimentação de velocidade convertida para milímetros por segundo.
    actualVelocityMmps : LREAL;

    // EN: Velocity reference accepted after inversion and equipment limiting.
    // PT: Referência de velocidade aceita após inversão e limitação do equipamento.
    commandedVelocityMmps : LREAL;

    // EN: One-cycle confirmation pulse after a position capture is accepted.
    // PT: Pulso de confirmação de um ciclo após uma captura de posição ser aceita.
    positionSetDone : BOOL;

    // EN: One-cycle indication that a position capture request was rejected.
    // PT: Indicação de um ciclo de que uma solicitação de captura de posição foi rejeitada.
    positionSetRejected : BOOL;

    // EN: Active position offset for commissioning and diagnostics.
    // PT: Offset de posição ativo para comissionamento e diagnóstico.
    positionOffsetMm : LREAL;
END_VAR

VAR
    // EN: Internal communication validation result.
    // PT: Resultado interno da validação da comunicação.
    communicationOkInternal : BOOL;

    // EN: Internal CiA 402 state decoded from the status word.
    // PT: Estado interno CiA 402 decodificado a partir da palavra de estado.
    deviceStateInternal : E_IS620P_CO_STATE;

    // EN: Internal validation of scaling parameters.
    // PT: Validação interna dos parâmetros de escala.
    configurationValidInternal : BOOL;

    // EN: Previous reset command state used for rising-edge detection.
    // PT: Estado anterior do comando de reset usado para detecção de borda de subida.
    resetFaultOld : BOOL;

    // EN: Rising edge of the fault reset command.
    // PT: Borda de subida do comando de reset de falha.
    resetFaultRisingEdge : BOOL;

    // EN: Previous zero-position command state used for rising-edge detection.
    // PT: Estado anterior do comando de zerar posição usado para detecção de borda de subida.
    zeroPositionOld : BOOL;

    // EN: Rising edge of the zero-position command.
    // PT: Borda de subida do comando de zerar posição.
    zeroPositionRisingEdge : BOOL;

    // EN: Previous set-position command state used for rising-edge detection.
    // PT: Estado anterior do comando de definir posição usado para detecção de borda de subida.
    setPositionOld : BOOL;

    // EN: Rising edge of the set-position command.
    // PT: Borda de subida do comando de definir posição.
    setPositionRisingEdge : BOOL;

    // EN: Indicates that the current position feedback can be calibrated.
    // PT: Indica que a realimentação de posição atual pode ser calibrada.
    positionSetAllowed : BOOL;

    // EN: Velocity reference limited in engineering units.
    // PT: Referência de velocidade limitada em unidades de engenharia.
    limitedVelocityMmps : LREAL;

    // EN: Raw velocity reference after conversion to drive units.
    // PT: Referência bruta de velocidade após conversão para unidades do drive.
    targetVelocityRaw : DINT;

    // EN: Timer reserved for the CiA 402 drive-enable sequence.
    // PT: Temporizador reservado para a sequência de habilitação CiA 402 do drive.
    enableTimer : TON;

    // EN: Timer reserved for operation-mode confirmation.
    // PT: Temporizador reservado para confirmação do modo de operação.
    modeSelectionTimer : TON;
END_VAR

// EN: Read and convert all hardware feedback before making control decisions.
// PT: Lê e converte todas as realimentações de hardware antes das decisões de controle.
_ReadHardwareInputs();

// EN: Decode the current CiA 402 state from the drive status word.
// PT: Decodifica o estado CiA 402 atual a partir da palavra de estado do drive.
deviceStateInternal := _DecodeDriveState(
    statusWordValue := HwToPlc.statusWord,
    communicationOk := communicationOkInternal
);

// EN: Process position calibration commands before publishing the current position.
// PT: Processa os comandos de calibração antes de publicar a posição atual.
_ProcessPositionCommands();

// EN: Generate the CiA 402 control word and operation-mode command.
// PT: Gera a palavra de controle CiA 402 e o comando do modo de operação.
_ControlDriveState();

// EN: Validate, limit and convert the velocity reference received from the parent block.
// PT: Valida, limita e converte a referência de velocidade recebida do bloco pai.
_ControlVelocity();

// EN: Publish the final generic device status at the end of the cycle.
// PT: Publica o estado genérico final do equipamento ao término do ciclo.
_UpdateStatus();

METHOD PRIVATE _ControlDriveState
// =============================================================================
// EN: Generates the CiA 402 control word and selects Profile Velocity mode.
// PT: Gera a palavra de controle CiA 402 e seleciona o modo Profile Velocity.
// =============================================================================
resetFaultRisingEdge := resetFault AND NOT resetFaultOld;
resetFaultOld := resetFault;

// EN: Keep mapped but unused profile-position references at safe values.
// PT: Mantém as referências mapeadas, porém não utilizadas, em valores seguros.
PlcToHw.targetPosition := 0;
PlcToHw.profileVelocity := 0;
PlcToHw.profileAcceleration := deviceConfig.profileAccelerationRaw;
PlcToHw.profileDeceleration := deviceConfig.profileDecelerationRaw;

IF enable THEN
    PlcToHw.modeCommand := 3;
ELSE
    PlcToHw.modeCommand := 0;
END_IF;

// EN: Monitor enable and mode-selection sequences without overriding the device state.
// PT: Monitora as sequências de habilitação e seleção de modo sem sobrescrever o estado do equipamento.
enableTimer(
    IN := enable AND enableDrive AND communicationOkInternal AND
          (deviceStateInternal <> E_IS620P_CO_STATE.OperationEnabled),
    PT := deviceConfig.enableTimeout
);

modeSelectionTimer(
    IN := enable AND enableDrive AND communicationOkInternal AND
          (HwToPlc.modeDisplay <> 3),
    PT := deviceConfig.modeSelectionTimeout
);

// EN: Priority: disabled, communication/configuration fault, quick stop, fault reset, normal state sequence.
// PT: Prioridade: desabilitado, falha de comunicação/configuração, quick stop, reset e sequência normal.
IF NOT enable THEN
    PlcToHw.controlWord := 16#0000;
ELSIF NOT communicationOkInternal OR NOT configurationValidInternal THEN
    PlcToHw.controlWord := 16#0000;
ELSIF quickStop THEN
    PlcToHw.controlWord := 16#0002;
ELSIF deviceStateInternal = E_IS620P_CO_STATE.Fault THEN
    IF resetFaultRisingEdge THEN
        PlcToHw.controlWord := 16#0080;
    ELSE
        PlcToHw.controlWord := 16#0000;
    END_IF;
ELSIF NOT enableDrive THEN
    PlcToHw.controlWord := 16#0006;
ELSE
    CASE deviceStateInternal OF
        E_IS620P_CO_STATE.SwitchOnDisabled:
            PlcToHw.controlWord := 16#0006;

        E_IS620P_CO_STATE.ReadyToSwitchOn:
            PlcToHw.controlWord := 16#0007;

        E_IS620P_CO_STATE.SwitchedOn,
        E_IS620P_CO_STATE.OperationEnabled,
        E_IS620P_CO_STATE.QuickStopActive:
            PlcToHw.controlWord := 16#000F;

        ELSE
            PlcToHw.controlWord := 16#0000;
    END_CASE;
END_IF;
END_METHOD

METHOD PRIVATE _ControlVelocity
// =============================================================================
// EN: Limits and converts the external velocity reference without generating a motion ramp.
// PT: Limita e converte a referência externa de velocidade sem gerar uma rampa de movimento.
// =============================================================================
limitedVelocityMmps := 0.0;
targetVelocityRaw := 0;
commandedVelocityMmps := 0.0;
PlcToHw.targetVelocity := 0;

IF enable AND
   enableDrive AND
   communicationOkInternal AND
   configurationValidInternal AND
   NOT quickStop AND
   (deviceStateInternal = E_IS620P_CO_STATE.OperationEnabled) AND
   (HwToPlc.modeDisplay = 3) THEN

    limitedVelocityMmps := LIMIT(
        -ABS(deviceConfig.maximumVelocityMmps),
        velocityReferenceMmps,
        ABS(deviceConfig.maximumVelocityMmps)
    );

    commandedVelocityMmps := limitedVelocityMmps;
    targetVelocityRaw := _ConvertVelocityToRaw(velocityMmps := limitedVelocityMmps);
    PlcToHw.targetVelocity := targetVelocityRaw;
END_IF;
END_METHOD

METHOD PRIVATE _ConvertRawPositionToMm : LREAL
// =============================================================================
// EN: Converts raw position feedback to millimeters without applying the calibration offset.
// PT: Converte a posição bruta para milímetros sem aplicar o offset de calibração.
// =============================================================================
VAR_INPUT
    rawPositionValue : DINT;
END_VAR
VAR
    convertedPositionMm : LREAL;
END_VAR
IF deviceConfig.positionUnitsPerMm <= 0.0 THEN
    _ConvertRawPositionToMm := 0.0;
    RETURN;
END_IF;

convertedPositionMm :=
    DINT_TO_LREAL(rawPositionValue) * deviceConfig.positionUnitsPerMm;

IF deviceConfig.directionInverted THEN
    convertedPositionMm := -convertedPositionMm;
END_IF;

_ConvertRawPositionToMm := convertedPositionMm;
END_METHOD

METHOD PRIVATE _ConvertRawVelocityToMmps : LREAL
// =============================================================================
// EN: Converts raw velocity feedback to millimeters per second.
// PT: Converte a velocidade bruta para milímetros por segundo.
// =============================================================================
VAR_INPUT
    rawVelocityValue : DINT;
END_VAR
VAR
    convertedVelocityMmps : LREAL;
END_VAR
IF deviceConfig.velocityUnitsPerMmps <= 0.0 THEN
    _ConvertRawVelocityToMmps := 0.0;
    RETURN;
END_IF;

convertedVelocityMmps :=
    DINT_TO_LREAL(rawVelocityValue) / deviceConfig.velocityUnitsPerMmps;

IF deviceConfig.directionInverted THEN
    convertedVelocityMmps := -convertedVelocityMmps;
END_IF;

_ConvertRawVelocityToMmps := convertedVelocityMmps;
END_METHOD

METHOD PRIVATE _ConvertVelocityToRaw : DINT
// =============================================================================
// EN: Converts a velocity command in millimeters per second to the signed raw drive value.
// PT: Converte um comando em milímetros por segundo para o valor bruto com sinal do drive.
// =============================================================================
VAR_INPUT
    velocityMmps : LREAL;
END_VAR
VAR
    driveVelocityMmps : LREAL;
    rawVelocityLreal  : LREAL;
END_VAR
IF deviceConfig.velocityUnitsPerMmps <= 0.0 THEN
    _ConvertVelocityToRaw := 0;
    RETURN;
END_IF;

driveVelocityMmps := velocityMmps;
IF deviceConfig.directionInverted THEN
    driveVelocityMmps := -driveVelocityMmps;
END_IF;

rawVelocityLreal := driveVelocityMmps * deviceConfig.velocityUnitsPerMmps;

IF rawVelocityLreal > 2147483647.0 THEN
    _ConvertVelocityToRaw := 2147483647;
ELSIF rawVelocityLreal < -2147483648.0 THEN
    _ConvertVelocityToRaw := -2147483647 - 1;
ELSE
    _ConvertVelocityToRaw := LREAL_TO_DINT(rawVelocityLreal);
END_IF;
END_METHOD

METHOD PRIVATE _DecodeDriveState : E_IS620P_CO_STATE
// =============================================================================
// EN: Decodes the CiA 402 Power Drive System state using the standard masks.
// PT: Decodifica o estado CiA 402 Power Drive System usando as máscaras padrão.
// =============================================================================
VAR_INPUT
    statusWordValue : UINT;
    communicationOk : BOOL;
END_VAR
VAR
    maskedState004F : UINT;
    maskedState006F : UINT;
END_VAR
IF NOT communicationOk THEN
    _DecodeDriveState := E_IS620P_CO_STATE.CommunicationFault;
    RETURN;
END_IF;

maskedState004F := statusWordValue AND 16#004F;
maskedState006F := statusWordValue AND 16#006F;

IF maskedState004F = 16#0000 THEN
    _DecodeDriveState := E_IS620P_CO_STATE.NotReadyToSwitchOn;
ELSIF maskedState004F = 16#0040 THEN
    _DecodeDriveState := E_IS620P_CO_STATE.SwitchOnDisabled;
ELSIF maskedState006F = 16#0021 THEN
    _DecodeDriveState := E_IS620P_CO_STATE.ReadyToSwitchOn;
ELSIF maskedState006F = 16#0023 THEN
    _DecodeDriveState := E_IS620P_CO_STATE.SwitchedOn;
ELSIF maskedState006F = 16#0027 THEN
    _DecodeDriveState := E_IS620P_CO_STATE.OperationEnabled;
ELSIF maskedState006F = 16#0007 THEN
    _DecodeDriveState := E_IS620P_CO_STATE.QuickStopActive;
ELSIF maskedState004F = 16#000F THEN
    _DecodeDriveState := E_IS620P_CO_STATE.FaultReactionActive;
ELSIF maskedState004F = 16#0008 THEN
    _DecodeDriveState := E_IS620P_CO_STATE.Fault;
ELSE
    _DecodeDriveState := E_IS620P_CO_STATE.NotReadyToSwitchOn;
END_IF;
END_METHOD

METHOD PRIVATE _ProcessPositionCommands
// =============================================================================
// EN: Captures a zero or an assigned engineering position by changing the persistent offset.
// PT: Captura zero ou uma posição de engenharia definida alterando o offset persistente.
// =============================================================================
positionSetDone := FALSE;
positionSetRejected := FALSE;

zeroPositionRisingEdge := zeroPosition AND NOT zeroPositionOld;
setPositionRisingEdge := setPosition AND NOT setPositionOld;

positionSetAllowed :=
    communicationOkInternal AND
    configurationValidInternal AND
    (ABS(actualVelocityMmps) <= ABS(deviceConfig.positionSetMaxVelocityMmps));

// EN: ZeroPosition has priority when both commands arrive in the same PLC cycle.
// PT: ZeroPosition possui prioridade quando ambos os comandos chegam no mesmo ciclo do PLC.
IF zeroPositionRisingEdge THEN
    IF positionSetAllowed THEN
        deviceConfig.positionOffsetMm := -rawPositionMm;
        deviceConfig.calibrationValid := TRUE;
        positionSetDone := TRUE;
    ELSE
        positionSetRejected := TRUE;
    END_IF;
ELSIF setPositionRisingEdge THEN
    IF positionSetAllowed THEN
        deviceConfig.positionOffsetMm := desiredPositionMm - rawPositionMm;
        deviceConfig.calibrationValid := TRUE;
        positionSetDone := TRUE;
    ELSE
        positionSetRejected := TRUE;
    END_IF;
END_IF;

zeroPositionOld := zeroPosition;
setPositionOld := setPosition;

// EN: Recalculate the published position immediately after an accepted capture.
// PT: Recalcula a posição publicada imediatamente após uma captura aceita.
actualPositionMm := rawPositionMm + deviceConfig.positionOffsetMm;
positionOffsetMm := deviceConfig.positionOffsetMm;
END_METHOD

METHOD PRIVATE _ReadHardwareInputs
// =============================================================================
// EN: Reads communication information and converts position and velocity feedback.
// PT: Lê as informações de comunicação e converte as realimentações de posição e velocidade.
// =============================================================================
// EN: NodeState 0 means no error. Value 64 also represents completed startup without a base error.
// PT: NodeState 0 significa sem erro. O valor 64 também representa startup concluído sem erro base.
communicationOkInternal := (HwToPlc.nodeState = 0) OR (HwToPlc.nodeState = 64);

// EN: Both conversion factors must be positive before motion references are accepted.
// PT: Ambos os fatores de conversão devem ser positivos antes de aceitar referências de movimento.
configurationValidInternal :=
    (deviceConfig.positionUnitsPerMm > 0.0) AND
    (deviceConfig.velocityUnitsPerMmps > 0.0) AND
    (deviceConfig.maximumVelocityMmps >= 0.0);

rawPosition := HwToPlc.actualPosition;
rawVelocity := HwToPlc.actualVelocity;

rawPositionMm := _ConvertRawPositionToMm(rawPositionValue := rawPosition);
actualPositionMm := rawPositionMm + deviceConfig.positionOffsetMm;
actualVelocityMmps := _ConvertRawVelocityToMmps(rawVelocityValue := rawVelocity);
positionOffsetMm := deviceConfig.positionOffsetMm;
END_METHOD

METHOD PRIVATE _UpdateStatus
// =============================================================================
// EN: Publishes communication, configuration and CiA 402 state information.
// PT: Publica informações de comunicação, configuração e estado CiA 402.
// =============================================================================
status.communicationOk := communicationOkInternal;
status.configurationValid := configurationValidInternal;
status.ready :=
    communicationOkInternal AND
    configurationValidInternal AND
    (deviceStateInternal = E_IS620P_CO_STATE.OperationEnabled) AND
    (HwToPlc.modeDisplay = 3);
status.driveEnabled := deviceStateInternal = E_IS620P_CO_STATE.OperationEnabled;
status.quickStopActive := deviceStateInternal = E_IS620P_CO_STATE.QuickStopActive;
status.calibrated := deviceConfig.calibrationValid;
status.warning := (HwToPlc.statusWord AND 16#0080) <> 0;
status.fault :=
    (deviceStateInternal = E_IS620P_CO_STATE.Fault) OR
    (deviceStateInternal = E_IS620P_CO_STATE.FaultReactionActive);
status.enableTimeout := enableTimer.Q;
status.modeSelectionTimeout := modeSelectionTimer.Q;
status.nodeState := HwToPlc.nodeState;
status.diagnosticFlag := HwToPlc.diagFlag;
status.statusWord := HwToPlc.statusWord;
status.activeMode := HwToPlc.modeDisplay;
status.deviceState := deviceStateInternal;
END_METHOD

END_FUNCTION_BLOCK

// ---- Library/EL6910 - TwinSAFE PLC/FB_EL6910.TcPOU
FUNCTION_BLOCK FB_EL6910
VAR_INPUT
	
		errorAcknowledgement : BOOL;
		run  : BOOL;
		safetyReset : BOOL;

END_VAR
VAR_OUTPUT

	eStop1Status	: EL6910_ESTOP_STATUS;
	eStop1Diagnostics : EL6910_ESTOP_DIGNOSTICS;

	eStop2Status	: EL6910_ESTOP_STATUS;
	eStop2Diagnostics : EL6910_ESTOP_DIGNOSTICS;

	eStop3Status	: EL6910_ESTOP_STATUS;
	eStop3Diagnostics : EL6910_ESTOP_DIGNOSTICS;

	eStop4Status	: EL6910_ESTOP_STATUS;
	eStop4Diagnostics : EL6910_ESTOP_DIGNOSTICS;
	

END_VAR
VAR
	    PDOS : EL6910_PDOS; // Process Data Objects for EL6910 communication
		EStop1DiagOld: INT;
		EStop2DiagOld: INT;
		EStop3DiagOld: INT;
		EStop4DiagOld: INT;

		
		
END_VAR


_eStopDiagnostics();
_eStopStatus();
_SafetyPLC();

METHOD PRIVATE _eStopDiagnostics
VAR_INPUT
END_VAR
//==============================================================
// E-STOP 1
//==============================================================

eStop1Diagnostics.discrepancyErrGroup1       := PDOS.HwToPLC.EStop1Diag.0;
eStop1Diagnostics.discrepancyErrGroup2       := PDOS.HwToPLC.EStop1Diag.1;
eStop1Diagnostics.discrepancyErrGroup3       := PDOS.HwToPLC.EStop1Diag.2;
eStop1Diagnostics.discrepancyErrGroup4       := PDOS.HwToPLC.EStop1Diag.3;

eStop1Diagnostics.edmMonitoringErr1          := PDOS.HwToPLC.EStop1Diag.4;
eStop1Diagnostics.edmMonitoringErr2          := PDOS.HwToPLC.EStop1Diag.5;

// Bits 6 and 7 are skipped (not used)

eStop1Diagnostics.discrepancyErrGroup1_Safe  := PDOS.HwToPLC.EStop1Diag.8;
eStop1Diagnostics.discrepancyErrGroup2_Safe  := PDOS.HwToPLC.EStop1Diag.9;
eStop1Diagnostics.discrepancyErrGroup3_Safe  := PDOS.HwToPLC.EStop1Diag.10;
eStop1Diagnostics.discrepancyErrGroup4_Safe  := PDOS.HwToPLC.EStop1Diag.11;


//==============================================================
// E-STOP 2
//==============================================================
eStop2Diagnostics.discrepancyErrGroup1       := PDOS.HwToPLC.EStop2Diag.0;
eStop2Diagnostics.discrepancyErrGroup2       := PDOS.HwToPLC.EStop2Diag.1;
eStop2Diagnostics.discrepancyErrGroup3       := PDOS.HwToPLC.EStop2Diag.2;
eStop2Diagnostics.discrepancyErrGroup4       := PDOS.HwToPLC.EStop2Diag.3;

eStop2Diagnostics.edmMonitoringErr1          := PDOS.HwToPLC.EStop2Diag.4;
eStop2Diagnostics.edmMonitoringErr2          := PDOS.HwToPLC.EStop2Diag.5;

// Bits 6 and 7 skipped (not used)

eStop2Diagnostics.discrepancyErrGroup1_Safe  := PDOS.HwToPLC.EStop2Diag.8;
eStop2Diagnostics.discrepancyErrGroup2_Safe  := PDOS.HwToPLC.EStop2Diag.9;
eStop2Diagnostics.discrepancyErrGroup3_Safe  := PDOS.HwToPLC.EStop2Diag.10;
eStop2Diagnostics.discrepancyErrGroup4_Safe  := PDOS.HwToPLC.EStop2Diag.11;


//==============================================================
// E-STOP 3
//==============================================================
eStop3Diagnostics.discrepancyErrGroup1       := PDOS.HwToPLC.EStop3Diag.0;
eStop3Diagnostics.discrepancyErrGroup2       := PDOS.HwToPLC.EStop3Diag.1;
eStop3Diagnostics.discrepancyErrGroup3       := PDOS.HwToPLC.EStop3Diag.2;
eStop3Diagnostics.discrepancyErrGroup4       := PDOS.HwToPLC.EStop3Diag.3;

eStop3Diagnostics.edmMonitoringErr1          := PDOS.HwToPLC.EStop3Diag.4;
eStop3Diagnostics.edmMonitoringErr2          := PDOS.HwToPLC.EStop3Diag.5;

// Bits 6 and 7 skipped (not used)

eStop3Diagnostics.discrepancyErrGroup1_Safe  := PDOS.HwToPLC.EStop3Diag.8;
eStop3Diagnostics.discrepancyErrGroup2_Safe  := PDOS.HwToPLC.EStop3Diag.9;
eStop3Diagnostics.discrepancyErrGroup3_Safe  := PDOS.HwToPLC.EStop3Diag.10;
eStop3Diagnostics.discrepancyErrGroup4_Safe  := PDOS.HwToPLC.EStop3Diag.11;


//==============================================================
// E-STOP 4
//==============================================================
eStop4Diagnostics.discrepancyErrGroup1       := PDOS.HwToPLC.EStop4Diag.0;
eStop4Diagnostics.discrepancyErrGroup2       := PDOS.HwToPLC.EStop4Diag.1;
eStop4Diagnostics.discrepancyErrGroup3       := PDOS.HwToPLC.EStop4Diag.2;
eStop4Diagnostics.discrepancyErrGroup4       := PDOS.HwToPLC.EStop4Diag.3;

eStop4Diagnostics.edmMonitoringErr1          := PDOS.HwToPLC.EStop4Diag.4;
eStop4Diagnostics.edmMonitoringErr2          := PDOS.HwToPLC.EStop4Diag.5;

// Bits 6 and 7 skipped (not used)

eStop4Diagnostics.discrepancyErrGroup1_Safe  := PDOS.HwToPLC.EStop4Diag.8;
eStop4Diagnostics.discrepancyErrGroup2_Safe  := PDOS.HwToPLC.EStop4Diag.9;
eStop4Diagnostics.discrepancyErrGroup3_Safe  := PDOS.HwToPLC.EStop4Diag.10;
eStop4Diagnostics.discrepancyErrGroup4_Safe  := PDOS.HwToPLC.EStop4Diag.11;
END_METHOD

METHOD PRIVATE _eStopStatus
VAR_INPUT
END_VAR


IF PDOS.HwToPLC.EStop1State <> EStop1DiagOld THEN
	
	// Reset all states to FALSE
	eStop1Status.estopState_RUN        := FALSE;
	eStop1Status.estopState_STOP       := FALSE;
	eStop1Status.estopState_SAFE       := FALSE;
	eStop1Status.estopState_ERROR      := FALSE;
	eStop1Status.estopState_RESET      := FALSE;
	eStop1Status.estopState_START      := FALSE;
	eStop1Status.estopState_DELAYOUT   := FALSE;

	CASE PDOS.HwToPLC.EStop1State OF
		
		1: eStop1Status.estopState_RUN        := TRUE;
		2: eStop1Status.estopState_STOP       := TRUE;
		3: eStop1Status.estopState_SAFE       := TRUE;
		4: eStop1Status.estopState_ERROR      := TRUE;
		5: eStop1Status.estopState_RESET      := TRUE;
		6: eStop1Status.estopState_START      := TRUE;
		8: eStop1Status.estopState_DELAYOUT   := TRUE;
	
	END_CASE
END_IF
	
EStop1DiagOld := PDOS.HwToPLC.EStop1State;


//==============================================================
// E-STOP 2
//==============================================================
IF PDOS.HwToPLC.EStop2State <> EStop2DiagOld THEN

    // Reset all states to FALSE
    eStop2Status.estopState_RUN       := FALSE;
    eStop2Status.estopState_STOP      := FALSE;
    eStop2Status.estopState_SAFE      := FALSE;
    eStop2Status.estopState_ERROR     := FALSE;
    eStop2Status.estopState_RESET     := FALSE;
    eStop2Status.estopState_START     := FALSE;
    eStop2Status.estopState_DELAYOUT  := FALSE;

    CASE PDOS.HwToPLC.EStop2State OF
        1: eStop2Status.estopState_RUN      := TRUE;
        2: eStop2Status.estopState_STOP     := TRUE;
        3: eStop2Status.estopState_SAFE     := TRUE;
        4: eStop2Status.estopState_ERROR    := TRUE;
        5: eStop2Status.estopState_RESET    := TRUE;
        6: eStop2Status.estopState_START    := TRUE;
        8: eStop2Status.estopState_DELAYOUT := TRUE;
    END_CASE
END_IF;

EStop2DiagOld := PDOS.HwToPLC.EStop2State;


//==============================================================
// E-STOP 3
//==============================================================
IF PDOS.HwToPLC.EStop3State <> EStop3DiagOld THEN

    // Reset all states to FALSE
    eStop3Status.estopState_RUN       := FALSE;
    eStop3Status.estopState_STOP      := FALSE;
    eStop3Status.estopState_SAFE      := FALSE;
    eStop3Status.estopState_ERROR     := FALSE;
    eStop3Status.estopState_RESET     := FALSE;
    eStop3Status.estopState_START     := FALSE;
    eStop3Status.estopState_DELAYOUT  := FALSE;

    CASE PDOS.HwToPLC.EStop3State OF
        1: eStop3Status.estopState_RUN      := TRUE;
        2: eStop3Status.estopState_STOP     := TRUE;
        3: eStop3Status.estopState_SAFE     := TRUE;
        4: eStop3Status.estopState_ERROR    := TRUE;
        5: eStop3Status.estopState_RESET    := TRUE;
        6: eStop3Status.estopState_START    := TRUE;
        8: eStop3Status.estopState_DELAYOUT := TRUE;
    END_CASE
END_IF;

EStop3DiagOld := PDOS.HwToPLC.EStop3State;


//==============================================================
// E-STOP 4
//==============================================================
IF PDOS.HwToPLC.EStop4State <> EStop4DiagOld THEN

    // Reset all states to FALSE
    eStop4Status.estopState_RUN       := FALSE;
    eStop4Status.estopState_STOP      := FALSE;
    eStop4Status.estopState_SAFE      := FALSE;
    eStop4Status.estopState_ERROR     := FALSE;
    eStop4Status.estopState_RESET     := FALSE;
    eStop4Status.estopState_START     := FALSE;
    eStop4Status.estopState_DELAYOUT  := FALSE;

    CASE PDOS.HwToPLC.EStop4State OF
        1: eStop4Status.estopState_RUN      := TRUE;
        2: eStop4Status.estopState_STOP     := TRUE;
        3: eStop4Status.estopState_SAFE     := TRUE;
        4: eStop4Status.estopState_ERROR    := TRUE;
        5: eStop4Status.estopState_RESET    := TRUE;
        6: eStop4Status.estopState_START    := TRUE;
        8: eStop4Status.estopState_DELAYOUT := TRUE;
    END_CASE
END_IF;

EStop4DiagOld := PDOS.HwToPLC.EStop4State;
END_METHOD

METHOD PRIVATE _SafetyPLC
VAR_INPUT
END_VAR

PDOS.PlcToHw.Run := run;
PDOS.PlcToHw.safetyReset := safetyReset;

PDOS.PlcToHw.ErrorAcknowledgement := errorAcknowledgement;
END_METHOD

END_FUNCTION_BLOCK

// ---- Library/Beckhoff/EL1008/FB_EL1008.TcPOU
FUNCTION_BLOCK FB_EL1008
VAR_INPUT
    // EN: Input forcing configuration used for commissioning.
    // PT: Configuração de force das entradas usada no comissionamento.
    deviceConfig : EL1008_DEV_CONFIG;
END_VAR

VAR_OUTPUT
    digitalInput_01 : BOOL;
    digitalInput_02 : BOOL;
    digitalInput_03 : BOOL;
    digitalInput_04 : BOOL;
    digitalInput_05 : BOOL;
    digitalInput_06 : BOOL;
    digitalInput_07 : BOOL;
    digitalInput_08 : BOOL;
END_VAR

VAR
    // EN: Process data mapped directly to the EL1008 input PDOs.
    // PT: Dados de processo mapeados diretamente nos PDOs de entrada do EL1008.
    PDOS : EL1008_HWTOPLC_PDOS;
END_VAR

inputState();

METHOD PRIVATE inputState
// EN: Map physical inputs and optional forced states to public outputs.
// PT: Mapeia as entradas físicas e os estados forçados opcionais para as saídas públicas.
digitalInput_01 := PDOS.digitalInput_00 OR (deviceConfig.enableForce AND deviceConfig.forceDigitalInput_00);
digitalInput_02 := PDOS.digitalInput_01 OR (deviceConfig.enableForce AND deviceConfig.forceDigitalInput_01);
digitalInput_03 := PDOS.digitalInput_02 OR (deviceConfig.enableForce AND deviceConfig.forceDigitalInput_02);
digitalInput_04 := PDOS.digitalInput_03 OR (deviceConfig.enableForce AND deviceConfig.forceDigitalInput_03);
digitalInput_05 := PDOS.digitalInput_04 OR (deviceConfig.enableForce AND deviceConfig.forceDigitalInput_04);
digitalInput_06 := PDOS.digitalInput_05 OR (deviceConfig.enableForce AND deviceConfig.forceDigitalInput_05);
digitalInput_07 := PDOS.digitalInput_06 OR (deviceConfig.enableForce AND deviceConfig.forceDigitalInput_06);
digitalInput_08 := PDOS.digitalInput_07 OR (deviceConfig.enableForce AND deviceConfig.forceDigitalInput_07);
END_METHOD

END_FUNCTION_BLOCK

// ---- Library/AxisControl/FB_ComplexAxisControl.TcPOU
FUNCTION_BLOCK FB_ComplexAxisControl
VAR_INPUT 
	
      enable                                     : Bool   := FALSE;                        // TRUE: Enable functionality of FB
      enableAxis                                 : Bool   := FALSE;                        // TRUE: Set axis enable; FALSE: Remove axis enable
      resetAxis                                  : Bool   := FALSE;                        // Rising edge: Acknowledgement of technology alarms or restart of the axis (depending on configuration)
      jogForward                                 : Bool   := FALSE;                        // Rising edge: Move an axis in jog mode (forward); Falling edge: Stop jogging
      jogBackward                                : Bool   := FALSE;                        // Rising edge: Move an axis in jog mode (backward); Falling edge: Stop jogging
      moveVelocity                               : Bool   := FALSE;                        // Rising edge: Move an axis at constant velocity/speed
      stop                                       : Bool   := FALSE;                        // Rising edge: Brake an axis until it comes to a standstill
      fastStop                                   : Bool   := FALSE;                        // Rising edge: Brake an axis until it comes to a standstill (with fastStop dynamics)
      torqueLimiting                             : Bool   := FALSE;                        // TRUE: Enable force/torque limiting
      homing                                     : Bool   := FALSE;                        // Rising edge: Home axis
	  homingSensor 								 : BOOL   := FALSE;                        // Rising edge: Home sensor input singnal
	  posRelative                                : BOOL   := FALSE;                        // Rising edge: Move an axis relative to its position when execution of the job began
      posAbsolute                                : Bool   := FALSE;                        // Rising edge: Move an axis to an absolute position
      posSuperimposed                            : Bool   := FALSE;                        // Rising edge: Start a superimposed positioning
      gearInRelative                             : Bool   := FALSE;                        // Rising edge: Start a gearing operation (relative)
      gearInAbsolute                             : Bool   := FALSE;                        // Rising edge: Start a gearing operation (absolute)
      camIn                                      : Bool   := FALSE;                        // Rising edge: Start a camming operation
      phasing                                    : Bool   := FALSE;                        // Rising edge: Start a phasing operation

   END_VAR

   VAR_OUTPUT 
	   
      valid                                      : Bool   := FALSE;                        // TRUE: Valid set of output values available at the FB
      busy                                       : Bool   := FALSE;                        // TRUE: FB is working and new output values can be expected
      error                                      : Bool   := FALSE;                        // TRUE: An error occurred while processing the FB
      status                                     : Word   := STATUS_NO_CALL;              // Current status of FB
      axisEnabled                                : Bool   := FALSE;                        // TRUE: The technology object is enabled. Motion commands can be executed
      resetActive                                : Bool   := FALSE;                        // TRUE: Reset/Restart of the axis is active
      commandBusy                                : Bool   := FALSE;                        // TRUE: The selected basic motion command is being executed
      commandDone                                : Bool   := FALSE;                        // TRUE: The selected basic motion command has completed without error
      commandAborted                             : Bool   := FALSE;                        // TRUE: The selected basic motion command has been aborted
      inVelocity                                 : Bool   := FALSE;                        // TRUE: The setpoint velocity/speed was reached and will be maintained
      inLimitation                               : Bool   := FALSE;                        // TRUE: The drive is operating at the force/torque limit
      homingCommandBusy                          : Bool   := FALSE;                        // TRUE: Homing command is being executed
      homingCommandDone                          : Bool   := FALSE;                        // TRUE: Homing command has completed without error
      homingCommandAborted                       : Bool   := FALSE;                        // TRUE: Homing command has been aborted
      superimposedBusy                           : Bool   := FALSE;                        // TRUE: The selected superimposed motion command is being executed
      superimposedDone                           : Bool   := FALSE;                        // TRUE: The selected superimposed motion command  has completed without error
      superimposedAborted                        : Bool   := FALSE;                        // TRUE: The selected superimposed motion command has been aborted
      inClamping                                 : Bool   := FALSE;                        // TRUE: The drive is kept at the fixed stop (clamping), the axis position is within the positioning tolerance
      startSync                                  : Bool   := FALSE;                        // TRUE: The axis is synchronizing to the leading axis
      inSync                                     : Bool   := FALSE;                        // TRUE: The axis is synchronized to the leading axis
      inSimulation                               : Bool   := FALSE;                        // TRUE: Synchronous operation is being simulated
      jogSelected                                : Bool   := FALSE;                        // TRUE: Jogging is active
      moveVelocitySelected                       : Bool   := FALSE;                        // TRUE: Moving with constant velocity/speed is active
      stopSelected                               : Bool   := FALSE;                        // TRUE: Stopping is active
      fastStopSelected                           : Bool   := FALSE;                        // TRUE: Stopping is active (with fastStop dynamics)
      torqueLimitingSelected                     : Bool   := FALSE;                        // TRUE: Force/Torque limiting is active
      homingSelected                             : Bool   := FALSE;                        // TRUE: Homing is active
      posRelativeSelected                        : Bool   := FALSE;                        // TRUE: Relative positioning is active
      posAbsoluteSelected                        : Bool   := FALSE;                        // TRUE: Absolute positioning is active
      posSuperimposedSelected                    : Bool   := FALSE;                        // TRUE: Superimposed positioning is active
      gearInRelativeSelected                     : Bool   := FALSE;                        // TRUE: Relative gearing is active
      gearInAbsoluteSelected                     : Bool   := FALSE;                        // TRUE: Absolute gearing is active
      camInSelected                              : Bool   := FALSE;                        // TRUE: Camming is active
      phasingSelected                            : BOOL   := FALSE;                        // TRUE: Phasing is active
      diagnostics                                : LAxisCtrl_typeDiagnostics;            // Diagnostics structure
   END_VAR

   VAR_IN_OUT 
        
	  axis      								 : AXIS_REF;                       // Reference to axis to be controlled
	  master                 					 : AXIS_REF;                       // Reference to leading axis for synchronous motion
      configuration                              : LAxisCtrl_typeAxisConfig;             // Structure for parameters
	  
   END_VAR

   VAR 
      statErrorUserCleared                       : Bool   := FALSE;                        // Error occurred that can only be solved by user; rising edge at enable input necessary
      statErrorAutoCleared                       : Bool   := FALSE;                        // Error occurred that can be acknowledged by FB
      statStatus                                 : Word   := STATUS_NO_CALL;              // Internal variable for status
      statDiagnostics                            : LAxisCtrl_typeDiagnostics;            // Internal variable for diagnostics
      statEnableOld                              : Bool   := FALSE;                        // Old value of enable for edge detection
      statFBState                                : SInt   := AXIS_MOTION;                 // State of FB (function block state machine)
      statFirstCycleReset                        : Bool   := TRUE;                         // TRUE: First cycle of reset command
      statPowerErrorOld                          : Bool   := FALSE;                        // Old value of MC_Power.error
      statResetState                             : Int    := CMD_IDLE;                    // State of reset command
      statFirstCycleResetError                   : Bool   := FALSE;                        // TRUE: First cycle of error in reset command
      statExtendedCommand                        : DWord  := CMD_NO_SELECTION;            // Variable for requested extended command (e.g. resetAxis, torquelimiting, homing)
      statExtendedCommandOld                     : DWord  := CMD_NO_SELECTION;            // Old value of variable for requested extended command
      statEnableAxisOld                          : Bool   := FALSE;                        // Old value of enableAxis for edge detection
      statEmptyDiagnostics                       : LAxisCtrl_typeDiagnostics;            // Internal empty diagnostic structure
      statHomingOld                              : Bool   := FALSE;                        // Old value of variable for homing command input
      statFirstCycleHoming                       : Bool   := TRUE;                         // TRUE: First cycle in homing command
      statPassiveHomingState                     : DInt   := NO_HOMING_ACTIVE;            // Current selected passive homing mode
      statExeOfHoming                            : Int    := CMD_BUSY;                    // Current state of execution of homing command
      statBasicCommand                           : DWord  := CMD_NO_SELECTION;            // Variable for requested basic motion command
      statBasicCommandOld                        : DWord  := CMD_NO_SELECTION;            // Old value of variable for requested basic motion command
      statBasicMotionState                       : DInt   := NO_SELECTION;                // State of selected basic motion command
      statExeOfBasicMotion                       : Int    := CMD_BUSY;                    // State of execution of current state of basic motion
      statFirstCycleBasicMotion                  : Bool   := TRUE;                         // TRUE: First cycle in respective state fo basic motion functionality
      statApplicativeBasicMotionError            : Bool   := FALSE;                        // TRUE: applicative error occurred (e.g. invalid direction configured)
      statVelocityChangeOnTheFly                 : Bool   := FALSE;                        // Velocity change on the fly is active
      statVelocity                               : LReal  := 0.0;                          // Internal variable for velocity
      statAcceleration                           : LReal  := 0.0;                          // Internal variable for acceleration
      statAbortAcceleration                      : Bool   := FALSE;                        // FALSE: The current acceleration at the start of the job is reduced using the configured jerk. Afterwards, the deceleration builds up; TRUE: The acceleration is set to 0.0 at the start of the job, and the deceleration immediately builds up.
      statDeceleration                           : LReal  := 0.0;                          // Internal variable for deceleration
      statJerk                                   : LReal  := 0.0;                          // Internal variable for jerk
      statPositionControlled                     : Bool   := TRUE;                         // FALSE: Non position-controlled operation; TRUE: Position-controlled operation
      statFirstCycleDone                         : Bool   := FALSE;                        // TRUE: First cycle of done at fastStop
      statTorqueLimitingState                    : SInt   := NO_TORQUE_LIMITING_ACTIVE;   // Current executed state for torquelimiting functionality
      statTorqueLimitingErrorOld                 : Bool   := FALSE;                        // TRUE: Error at Torquelimiting occurred last cycle
      statTorqueLimit                            : LReal  := -1.0;                         // Value of force/torque limiting (in the configured unit of measurement)
      statJogMode                                : DInt   := JOG_MODE_CONTINUOUS;         // Current selected jog mode
      statDirection                              : Int    := SPECIFIED_DIR;               // Internal variable for direction of rotation of the axis
      statHomingPosition                         : LReal  := 0.0;                          // The specified value is used according to the selected "Mode".
      statHomingSubState                         : SInt   := HOMING_IDLE;                 // Current subState of execution of homing functionality
      statIncJogSubState                         : SInt   := INC_JOG_IDLE;                // Current subState of execution of jog incremental functionality
      statIncJogStartPosition                    : LReal  := 0.0;                          // Last stored axis position (for incremental jogging)
      statIncJogDirectionOld                     : Int    := 0;                            // Old value of direction of executing incremental jogging
      statIncrement                              : LReal  := 0.0;                          // Jog Incremental: distance of Increment (positive or negative)
      statIncJogDistance                         : LReal  := 0.0;                          // Jog Incremental: current distance to destination position
      statResetIncJog                            : Bool   := TRUE;                         // TRUE: First cycle in incremental jogging state (detection of new increment)
      statPosition                               : LReal  := 0.0;                          // Internal variable for position
      statPositionChangeOnTheFly                 : Bool   := FALSE;                        // Position change on the fly is active
      statHomingMode                             : Int    := DIRECT_HOMING;               // Operating Mode of MC_HOME command
      statActiveHomingState                      : DInt   := NO_HOMING_ACTIVE;            // Current selected active homing mode
      statSupImpCommand                          : DWord  := CMD_NO_SELECTION;            // Variable for requested superimposed motion command
      statSupImpCommandOld                       : DWord  := CMD_NO_SELECTION;            // Old value of variable for requested superimposed motion command
      statSupImpMotionState                      : DInt   := NO_SELECTION;                // Current selected superimposed motion functionality
      statExeOfSupImpMotionState                 : Int    := CMD_BUSY;                    // Current state of execution of superimposed basic motion
      statFirstCycleSupImpMotion                 : Bool   := TRUE;                         // TRUE: First cycle in positioning (superimposed) functionality
      statSupImpMotionPosition                   : LReal  := 0.0;                          // Position setpoint (for posSuperimposed command)
      statApplicativeSupImpMotionError           : Bool   := FALSE;                        // TRUE: applicative error occurred (e.g. invalid direction configured)
      statRatioChangeOnTheFly                    : Bool   := FALSE;                        // Ratio change on the fly is active
      statChangePhaseShiftOnTheFly               : Bool   := FALSE;                        // Phase shift change on the fly is active
      statPhaseShift                             : LReal  := 0.0;                          // Relative/Absolute master value shift
      statPhaseAbsolute                          : Bool   := TRUE;                         // Indicates the type of phase shift (TRUE: The phase shift is taken over as an absolute value; FALSE: The phase shift is added to an existing offset)
      statRatioNumerator                         : DInt   := 1;                            // Gear ratio numerator
      statRatioDenominator                       : DInt   := 1;                            // Gear ratio denominator
      statEnableAxis                             : Bool   := FALSE;                        // Internal variable for enabling axis
      statSyncMotionSimulationState              : SInt   := AXIS_NOT_IN_SIM;             // Current executed state for synchronized motion simulation
      statSynchronizedMotionErrorOld             : Bool   := FALSE;                        // Old value of MC_SynchronizedMotionSimulation.error
      statMainSelectionState                     : Int    := 0;                            // Current executed State for execution of basic motion commands or reset of waiting gearing / camming commands
      statMasterSyncPosition                     : LReal  := 0.0;                          // Synchronous position of leading axis. Position of the following axis starting from which the leading and following axes move synchronously
      statSlaveSyncPosition                      : LReal  := 0.0;                          // Synchronous position of leading axis. Position of the leading axis starting from which the leading and following axes move synchronously
      statSyncDirection                          : DInt   := FORWARD_DIR;                 // Direction of synchronization
      statMasterStartDistance                    : LReal  := 0.0;                          // Master value distance (when "SyncProfileReference" = 1)
      statSyncProfileReference                   : DInt   := 0;                            // Type of synchronization
      statApplicationMode                        : DInt   := 0;                            // Application of cam
      //statCam                                    : DB_ANY;                                 // Internal variable for cam
      instPower                                  : MC_POWER;                               // Instance of MC_Power
      instReset                                  : MC_RESET;                               // Instance of MC_Reset
      instHome                                   : MC_HOME;                                // Instance of MC_Home
      instHalt                                   : MC_HALT;                                // Instance of MC_Halt
      instMoveJog                                : MC_JOG;                             // Instance of MC_MoveJog
      instTorqueLimiting                         : MC_TORQUELIMITING;                      // Instance of MC_TorqueLimiting
      instMoveVelocity                           : MC_MOVEVELOCITY;                        // Instance of MC_MoveVelocity
      instMoveRelative                           : MC_MOVERELATIVE;                        // Instance of MC_MoveRelative
      instMoveAbsolute                           : MC_MOVEABSOLUTE;                        // Instance of MC_MoveAbsolute
      instMoveSuperimposed                       : MC_MOVESUPERIMPOSED;                    // Instance of MC_MoveSuperimposed
      instGearIn                                 : MC_GEARIN;                              // Instance of MC_GearIn
      instPhasingAbsolute                        : MC_PHASINGABSOLUTE;                     // Instance of MC_PhasingAbsolute
      instPhasingRelative                        : MC_PHASINGRELATIVE;                     // Instance of MC_PhasingRelative
      instGearInPos                              : MC_GEARINDYN;                           // Instance of MC_GearInPos
      instCamIn                                  : MC_CAMIN;                               // Instance of MC_CamIn
	//instAxisStatus							 : FB_AxisStatus;							// Instance of FB_AXIS_STATUS
	//instSyncMotionSimulation                   : MC_SYNCHRONIZEDMOTIONSIMULATION;        // Instance of MC_SynchronizedMotionSimulation
	  instTimerTON								 : TON;
	  StatusWord: INT;
	  
END_VAR
	  
	  VAR_TEMP
	  
	  tempNewExtendedCmd                         : DINT;                                   // Temporary variable for extended command
      tempEnableAxis                             : Bool;                                   // Temporary variable for enableAxis
      tempErrorInCmd                             : Bool;                                   // Temporary variable for error in actual command
      tempRisingCmd                              : DWord;                                  // Temporary DWord which indicates all rising edges of command word
      tempStopCmdSelected                        : Bool;                                   // TRUE: Stop or faststop selected in current cycle
      tempDword                                  : DWord;                                  // Temporary DWord for evaluation of rising edges of basic command word
      tempIndex                                  : Int;                                    // Temporary index
      tempCountRisEdges                          : USInt;                                  // Temporary counter for rising edges in command word
      tempNewBasicMotionCmd                      : DInt;                                   // Temporary variable for basic motion command
      tempStateChangeActive                      : Bool;                                   // TRUE: State change is active, stay in loop for one more cycle
      tempStatusWord                             : DWord;                                  // Temporary variable for statusword of axis
      tempNewSupImpCmd                           : DInt;                                   // Temporary variable for superimposed motion command
      tempHoming                                 : BOOL;                                   // Temporary variable for homing command
  	  tempFalse									 : BOOL;
   END_VAR

